FUNCTION_BLOCK FB_CHPSystem EXTENDS FB_SystemContinous
VAR_INPUT
END_VAR
VAR_OUTPUT
END_VAR
VAR
END_VAR

END_FUNCTION_BLOCK

(* stored: Version 1.1.0.1, ProductVersion 3.1.4024.10
   POU FB_CHPSystem: Id {03be9f87-4e59-4877-a478-dceefb67f1c9}, SpecialFunc None *)
